PROGRAM INTERNAL PRG_TESTS

(* Instantiate test suites here. Naming convention for tests should be a suffix with _Tests.
Good practice for creating test methods is to end them with _test as well. *)
VAR

	XV03ValveSystem_Tests		: FB_XV03ValveSystem_Tests;
	XV03DiagnosisParser_Tests	: FB_XV03_DiagnosticsParser;
END_VAR

// Run tests in paralel
// TcUnit.RUN();

// Run tests in sequence, one after the other. Uncomment if required.
TcUnit.RUN_IN_SEQUENCE();

END_PROGRAM

(* stored: Version 1.1.0.1, ProductVersion 3.1.4024.16
   POU PRG_TESTS: Id {f8808f06-636f-0b21-3e49-c04e8ee4c465}, SpecialFunc None *)
